FUNCTION_BLOCK PrintInt
  (* Standard: 61499-2 *)
  (* Version 0.1, 2017-00-09, hpea485, UOA *)
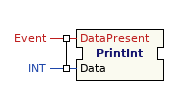
  EVENT_INPUT
    DataPresent WITH Data;
  END_EVENT
  VAR_INPUT
    Data : INT;
  END_VAR
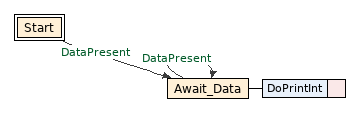
  EC_STATES
    Start;
    Await_Data : DoPrintInt;
  END_STATES
  EC_TRANSITIONS
    Start TO Await_Data := DataPresent;
    Await_Data TO Await_Data := DataPresent;
  END_TRANSITIONS
  ALGORITHM DoPrintInt IN C:
printf("PrintInt: %d\n", me->Data);
  END_ALGORITHM
END_FUNCTION_BLOCK
